{attribute addProperty BoxType "EL3453-0000-0018"}
{attribute addProperty Id "L1_StatusAT %I*L1_Status_EEFC181480100L1_BasicAT %I*L1_Basic_005DC40B6480L1_PowerAT %I*L1_Power_E8C64AA4128160L2_StatusAT %I*L2_Status_EEFC181480100L2_BasicAT %I*L2_Basic_005DC40B6480L2_PowerAT %I*L2_Power_E8C64AA4128160L3_StatusAT %I*L3_Status_EEFC181480100L3_BasicAT %I*L3_Basic_005DC40B6480L3_PowerAT %I*L3_Power_E8C64AA4128160Total_StatusAT %I*Total_Status_0C568DD4136170Total_BasicAT %I*Total_Basic_93D5BCB4160200WcStateAT %I*WcState_98A4DF7520.250InfoDataAT %I*InfoData_BC63D37F80100"}
{attribute addProperty CRC "3075133163"}
{attribute addProperty SizeInBites "1194"}
{attribute addProperty SizeInBytes "149.25"}
TYPE EL3453_BDDFEB0B :
STRUCT
	{attribute addProperty Name "L1_Status"}
	L1_Status : L1_Status_EEFC1814;
	{attribute addProperty Name "L1_Basic"}
	L1_Basic : L1_Basic_005DC40B;
	{attribute addProperty Name "L1_Power"}
	L1_Power : L1_Power_E8C64AA4;
	{attribute addProperty Name "L2_Status"}
	L2_Status : L2_Status_EEFC1814;
	{attribute addProperty Name "L2_Basic"}
	L2_Basic : L2_Basic_005DC40B;
	{attribute addProperty Name "L2_Power"}
	L2_Power : L2_Power_E8C64AA4;
	{attribute addProperty Name "L3_Status"}
	L3_Status : L3_Status_EEFC1814;
	{attribute addProperty Name "L3_Basic"}
	L3_Basic : L3_Basic_005DC40B;
	{attribute addProperty Name "L3_Power"}
	L3_Power : L3_Power_E8C64AA4;
	{attribute addProperty Name "Total_Status"}
	Total_Status : Total_Status_0C568DD4;
	{attribute addProperty Name "Total_Basic"}
	Total_Basic : Total_Basic_93D5BCB4;
	{attribute addProperty Name "WcState"}
	WcState : WcState_98A4DF75;
	{attribute addProperty Name "InfoData"}
	InfoData : InfoData_BC63D37F;
END_STRUCT
END_TYPE

(* stored: Version 1.2.0.0, ProductVersion 3.1.4024.9
   DUT EL3453_BDDFEB0B: Id {f1c7f489-18c2-4fcf-865d-dc88a113024b} *)
